TEXTLIST EL2809_M_1
  1 = 'F Pump1' | chinese: '清洗液泵1' | Chinese: '图层泵1'
  2 = 'F Pump2' | chinese: '清洗液泵2' | Chinese: '图层泵2'
  3 = 'W ink tank stirring_F' | chinese: '白墨瓶搅拌（正转）' | Chinese: '白墨瓶搅拌（正转）'
  4 = 'W ink tank stirring_B' | chinese: '白墨瓶搅拌（反转）' | Chinese: '白墨瓶搅拌（反转）'
  5 = 'LED_C' | chinese: '墨瓶C  LED' | Chinese: '墨瓶C  LED'
  6 = 'LED_Y' | chinese: '墨瓶Y  LED' | Chinese: '墨瓶Y  LED'
  7 = 'LED_M' | chinese: '墨瓶M  LED' | Chinese: '墨瓶M  LED'
  8 = 'LED_K' | chinese: '墨瓶K  LED' | Chinese: '墨瓶K  LED'
  9 = 'LED_LC' | chinese: '墨瓶LC  LED' | Chinese: '墨瓶LC  LED'
  10 = 'LED_LM' | chinese: '墨瓶LM  LED' | Chinese: '墨瓶LM  LED'
  11 = 'LED_P' | chinese: '墨瓶P LED' | Chinese: '墨瓶W  LED'
  12 = 'LED_W' | chinese: '墨瓶W LED' | Chinese: '墨瓶清洗液  LED'
  13 = 'LED_F' | chinese: '墨瓶F  LED' | Chinese: '墨瓶图层  LED'
  14 = 'LED_Waste' | chinese: '墨瓶废液  LED' | Chinese: '墨瓶废液  LED'
  15 = 'Waste liquid  fan' | chinese: '废液吸风扇' | Chinese: '废液吸风扇'
  16 = 'Waste Pump' | chinese: '废液泵' | Chinese: '废液泵'
   = ''
END_TEXTLIST

(* stored: Version 1.1.0.1, ProductVersion 3.1.4024.11
   TextList EL2809_M_1: Id {b0c12962-faf2-4936-ae6e-9637ae91af20} *)
